PROGRAM Circuito_L7
VAR_INPUT
	Modo_Calibrar_L7: BOOL;
END_VAR
VAR
		fbBomba_L7 :Equipo_Motor_ATV320;
		ControlValv_ioLink_V1:ControlValv_ioLink;
		ControlValv_ioLink_V2: ControlValv_ioLink;
		ControlValv_ioLink_V3: ControlValv_ioLink;
		ControlValv_ioLink_V4: ControlValv_ioLink;
		Falla_L7_V1:BOOL;
		Falla_L7_V2:BOOL;
		Falla_L7_V3:BOOL;
		Falla_L7_V4:BOOL;
	Balanza_PU2_WT7: Balanza;
		dHS:DINT;
		TOF_calibradoIBC: TOF;
		PID_L7_SP:REAL;
		PID_L7_auto:BOOL;
		PID_L7_reset:BOOL;
		PID_L7_manual:REAL;
		PID_L7_bMuerta:REAL := 5;
		PID_L7_Kp:REAL := 0.1;
		PID_L7_Ti:REAL := 100;
		PID_L7_PV:REAL;
		Dosis_L7	:REAL;
		TiempoInyeccion_L7	:DINT;
		Peso	:REAL;
		Offset_L7:REAL;
		Inyeccion_L7:BOOL;
		Volumen_L7:REAL;
		Calculo_caudal_L7: Calculo_caudal;
		CorrecionCaudalxOffset_L7: CorrecionCaudalxOffset;
		tInyeccion: TON;
		Total :REAL;
		Totalant	:REAL;
		auxIniCal:BOOL;
		AuxVol:REAL;
		CA2_L7_V1_CmdA_Man :BOOL;
		CA2_L7_V4_CmdA_Man :BOOL;
		TDemoraInyectar: TON;
		SetDemoraInyeccion: REAL;
		Tiempo_seg_to_TIME_DemoraInyec: Tiempo_seg_to_TIME;
		AuxTDemoraInyec: TIME;
		PID_L7: FB_PID;
		Tiempo_TIME_to_seg_InyCal: Tiempo_TIME_to_seg;
		AuxInyCal:TIME;		
		IniTotalFT2:REAL;
		Auxconsumo:REAL;	
	ProductoAsociado: STRING;
	Lavagem_Circuito07: Lavagem;
	Calibracao_teste: Calibracao_V03;
END_VAR

VAR PERSISTENT
	UltimaCalibracao	:UDINT;	//Data e hora da ultima calibração
END_VAR
VAR // added by the converter: edge detectors and wires of the graphical bodies
    _w1, _w2, _w3, _w4, _w5, _w6, _w7, _w8, _w9, _w10, _w11, _w12, _w13 : BOOL;
    _ft1 : F_TRIG;
    _rt1, _rt2 : R_TRIG;
END_VAR

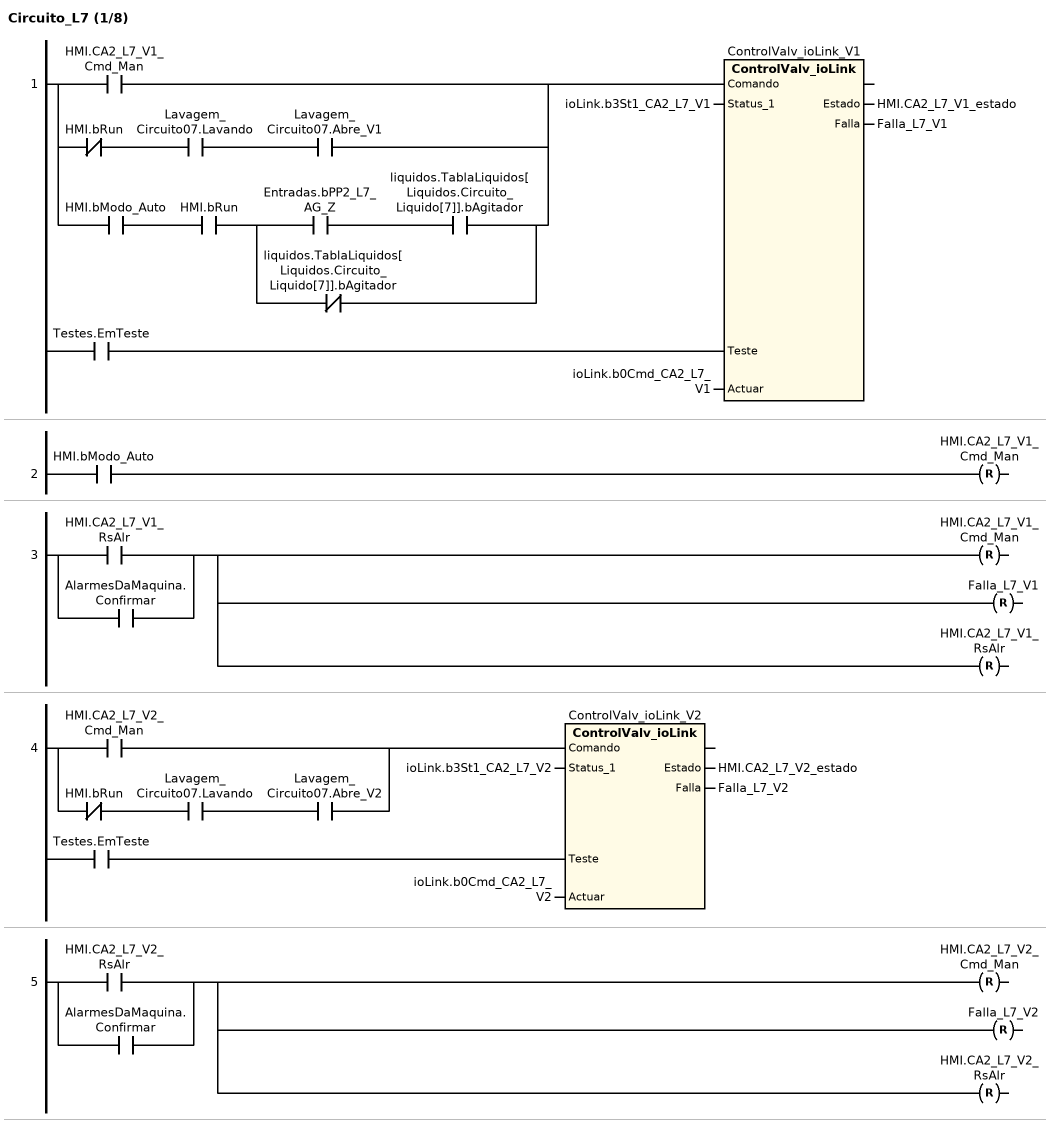
// NETWORK 1
ControlValv_ioLink_V1(
    Comando := HMI.CA2_L7_V1_Cmd_Man OR NOT HMI.bRun AND Lavagem_Circuito07.Lavando AND Lavagem_Circuito07.Abre_V1 OR HMI.bModo_Auto AND HMI.bRun AND (Entradas.bPP2_L7_AG_Z AND (liquidos.TablaLiquidos[Liquidos.Circuito_Liquido[7]].bAgitador) OR NOT (liquidos.TablaLiquidos[Liquidos.Circuito_Liquido[7]].bAgitador)),
    Status_1 := ioLink.b3St1_CA2_L7_V1,
    Teste := Testes.EmTeste,
    Actuar := ioLink.b0Cmd_CA2_L7_V1,
    Estado => HMI.CA2_L7_V1_estado,
    Falla => Falla_L7_V1); // ControlValv_ioLink

// NETWORK 2
HMI.CA2_L7_V1_Cmd_Man R= HMI.bModo_Auto;

// NETWORK 3
_w1 := HMI.CA2_L7_V1_RsAlr OR AlarmesDaMaquina.Confirmar;
HMI.CA2_L7_V1_Cmd_Man R= _w1;
Falla_L7_V1 R= _w1;
HMI.CA2_L7_V1_RsAlr R= _w1;

// NETWORK 4
ControlValv_ioLink_V2(
    Comando := HMI.CA2_L7_V2_Cmd_Man OR NOT HMI.bRun AND Lavagem_Circuito07.Lavando AND Lavagem_Circuito07.Abre_V2,
    Status_1 := ioLink.b3St1_CA2_L7_V2,
    Teste := Testes.EmTeste,
    Actuar := ioLink.b0Cmd_CA2_L7_V2,
    Estado => HMI.CA2_L7_V2_estado,
    Falla => Falla_L7_V2); // ControlValv_ioLink

// NETWORK 5
_w2 := HMI.CA2_L7_V2_RsAlr OR AlarmesDaMaquina.Confirmar;
HMI.CA2_L7_V2_Cmd_Man R= _w2;
Falla_L7_V2 R= _w2;
HMI.CA2_L7_V2_RsAlr R= _w2;

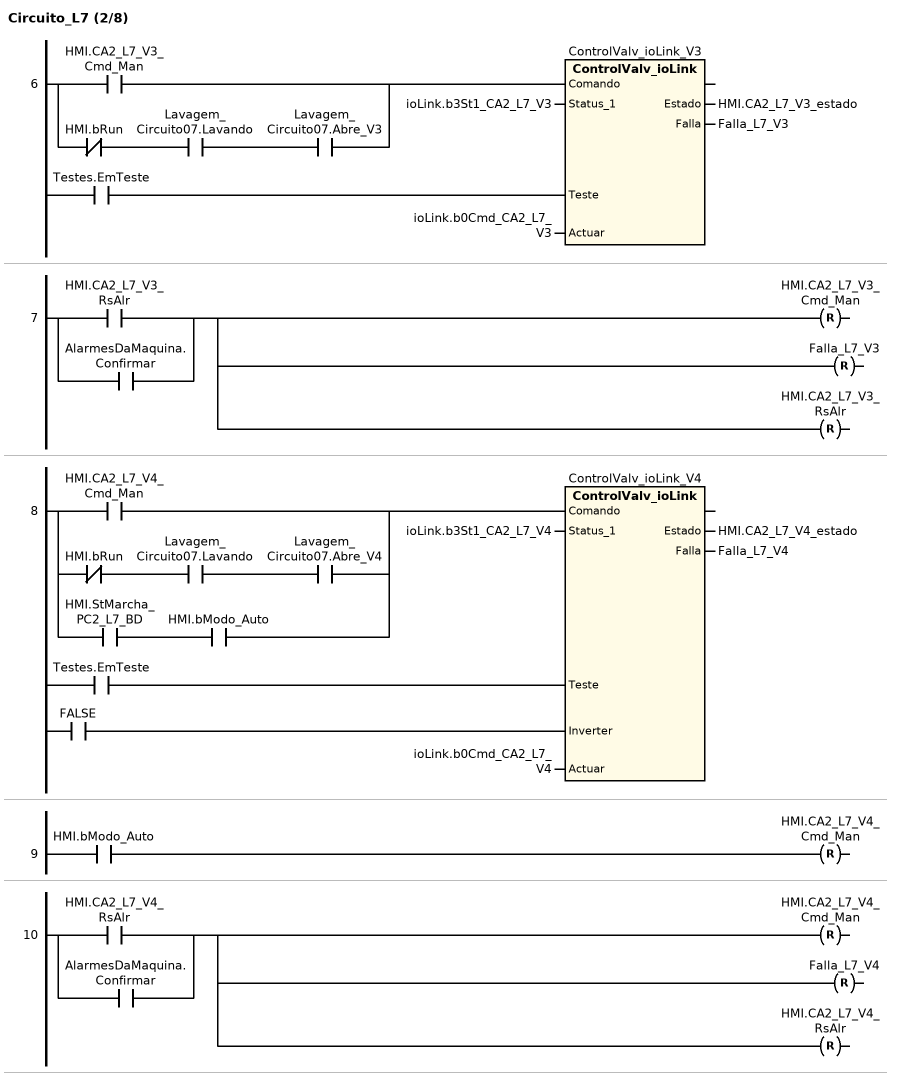
// NETWORK 6
ControlValv_ioLink_V3(
    Comando := HMI.CA2_L7_V3_Cmd_Man OR NOT HMI.bRun AND Lavagem_Circuito07.Lavando AND Lavagem_Circuito07.Abre_V3,
    Status_1 := ioLink.b3St1_CA2_L7_V3,
    Teste := Testes.EmTeste,
    Actuar := ioLink.b0Cmd_CA2_L7_V3,
    Estado => HMI.CA2_L7_V3_estado,
    Falla => Falla_L7_V3); // ControlValv_ioLink

// NETWORK 7
_w3 := HMI.CA2_L7_V3_RsAlr OR AlarmesDaMaquina.Confirmar;
HMI.CA2_L7_V3_Cmd_Man R= _w3;
Falla_L7_V3 R= _w3;
HMI.CA2_L7_V3_RsAlr R= _w3;

// NETWORK 8
ControlValv_ioLink_V4(
    Comando := HMI.CA2_L7_V4_Cmd_Man OR NOT HMI.bRun AND Lavagem_Circuito07.Lavando AND Lavagem_Circuito07.Abre_V4 OR HMI.StMarcha_PC2_L7_BD AND HMI.bModo_Auto,
    Status_1 := ioLink.b3St1_CA2_L7_V4,
    Teste := Testes.EmTeste,
    Inverter := FALSE,
    Actuar := ioLink.b0Cmd_CA2_L7_V4,
    Estado => HMI.CA2_L7_V4_estado,
    Falla => Falla_L7_V4); // ControlValv_ioLink

// NETWORK 9
HMI.CA2_L7_V4_Cmd_Man R= HMI.bModo_Auto;

// NETWORK 10
_w4 := HMI.CA2_L7_V4_RsAlr OR AlarmesDaMaquina.Confirmar;
HMI.CA2_L7_V4_Cmd_Man R= _w4;
Falla_L7_V4 R= _w4;
HMI.CA2_L7_V4_RsAlr R= _w4;

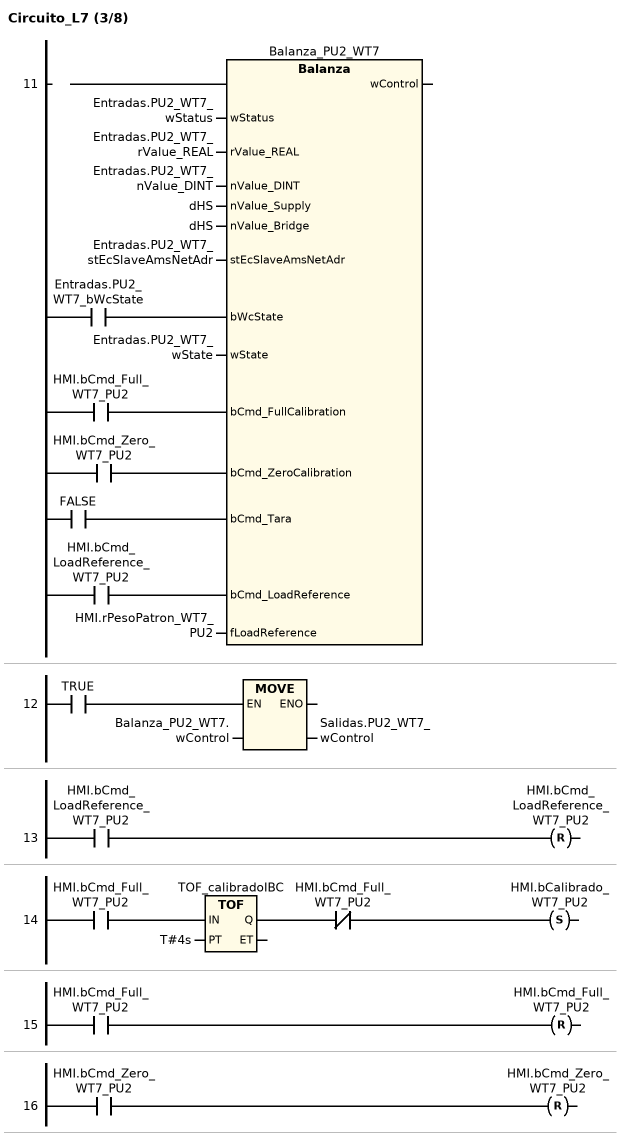
// NETWORK 11
Balanza_PU2_WT7(
    wStatus := Entradas.PU2_WT7_wStatus,
    rValue_REAL := Entradas.PU2_WT7_rValue_REAL,
    nValue_DINT := Entradas.PU2_WT7_nValue_DINT,
    nValue_Supply := dHS,
    nValue_Bridge := dHS,
    stEcSlaveAmsNetAdr := Entradas.PU2_WT7_stEcSlaveAmsNetAdr,
    bWcState := Entradas.PU2_WT7_bWcState,
    wState := Entradas.PU2_WT7_wState,
    bCmd_FullCalibration := HMI.bCmd_Full_WT7_PU2,
    bCmd_ZeroCalibration := HMI.bCmd_Zero_WT7_PU2,
    bCmd_Tara := FALSE,
    bCmd_LoadReference := HMI.bCmd_LoadReference_WT7_PU2,
    fLoadReference := HMI.rPesoPatron_WT7_PU2); // Balanza

// NETWORK 12
Salidas.PU2_WT7_wControl := Balanza_PU2_WT7.wControl;

// NETWORK 13
HMI.bCmd_LoadReference_WT7_PU2 R= HMI.bCmd_LoadReference_WT7_PU2;

// NETWORK 14
TOF_calibradoIBC(IN := HMI.bCmd_Full_WT7_PU2, PT := T#4s); // TOF
HMI.bCalibrado_WT7_PU2 S= TOF_calibradoIBC.Q AND NOT HMI.bCmd_Full_WT7_PU2;

// NETWORK 15
HMI.bCmd_Full_WT7_PU2 R= HMI.bCmd_Full_WT7_PU2;

// NETWORK 16
HMI.bCmd_Zero_WT7_PU2 R= HMI.bCmd_Zero_WT7_PU2;

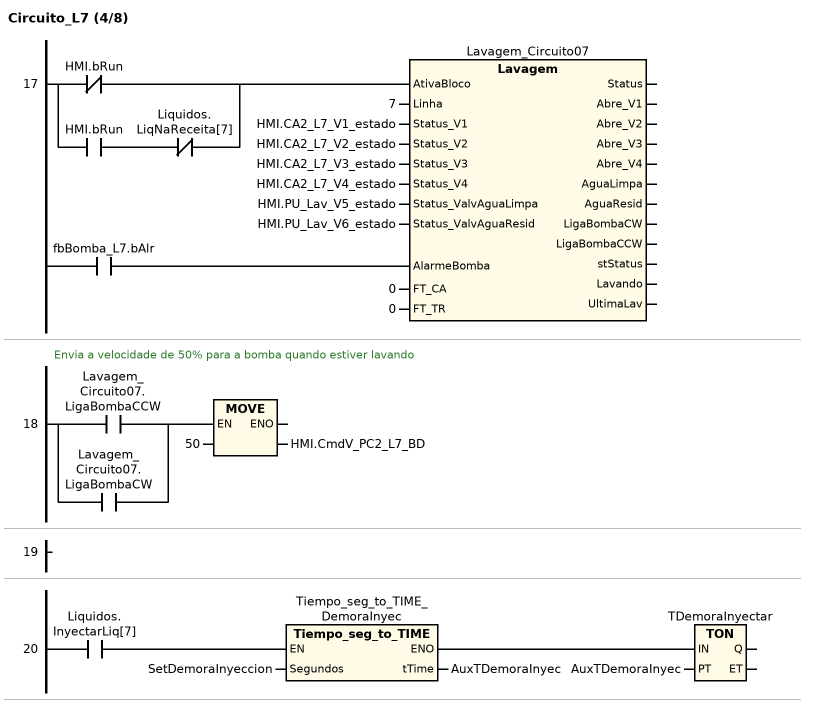
// NETWORK 17
Lavagem_Circuito07(
    AtivaBloco := NOT HMI.bRun OR HMI.bRun AND NOT Liquidos.LiqNaReceita[7],
    Linha := 7,
    Status_V1 := HMI.CA2_L7_V1_estado,
    Status_V2 := HMI.CA2_L7_V2_estado,
    Status_V3 := HMI.CA2_L7_V3_estado,
    Status_V4 := HMI.CA2_L7_V4_estado,
    Status_ValvAguaLimpa := HMI.PU_Lav_V5_estado,
    Status_ValvAguaResid := HMI.PU_Lav_V6_estado,
    AlarmeBomba := fbBomba_L7.bAlr,
    FT_CA := 0,
    FT_TR := 0); // Lavagem

// NETWORK 18
// Envia a velocidade de 50% para a bomba quando estiver lavando
IF Lavagem_Circuito07.LigaBombaCCW OR Lavagem_Circuito07.LigaBombaCW THEN HMI.CmdV_PC2_L7_BD := 50; END_IF

// NETWORK 19

// NETWORK 20
_w5 := Liquidos.InyectarLiq[7];
IF _w5 THEN
    Tiempo_seg_to_TIME_DemoraInyec(Segundos := SetDemoraInyeccion, tTime => AuxTDemoraInyec); // Tiempo_seg_to_TIME
END_IF
TDemoraInyectar(IN := _w5, PT := AuxTDemoraInyec); // TON

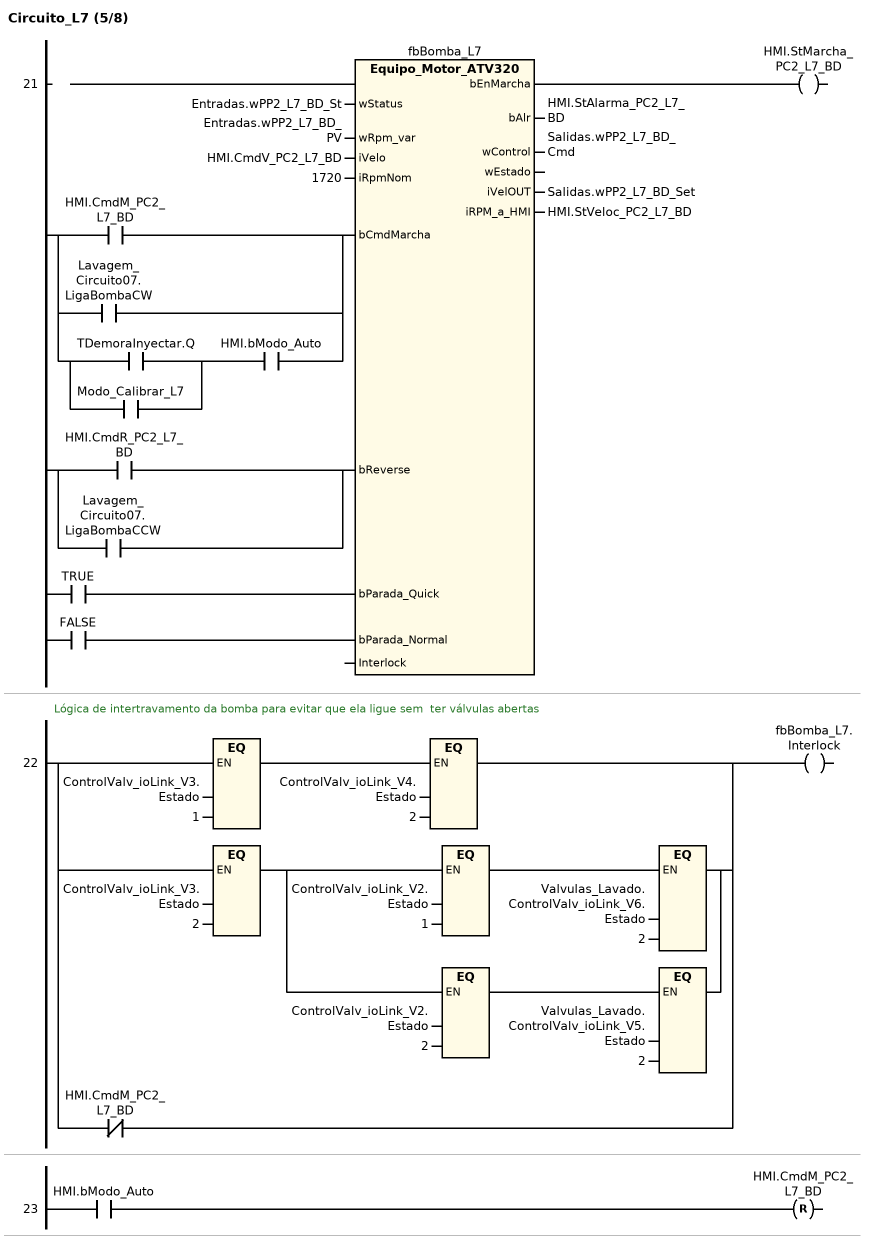
// NETWORK 21
fbBomba_L7(
    wStatus := Entradas.wPP2_L7_BD_St,
    wRpm_var := Entradas.wPP2_L7_BD_PV,
    iVelo := HMI.CmdV_PC2_L7_BD,
    iRpmNom := 1720,
    bCmdMarcha := HMI.CmdM_PC2_L7_BD OR Lavagem_Circuito07.LigaBombaCW OR (TDemoraInyectar.Q OR Modo_Calibrar_L7) AND HMI.bModo_Auto,
    bReverse := HMI.CmdR_PC2_L7_BD OR Lavagem_Circuito07.LigaBombaCCW,
    bParada_Quick := TRUE,
    bParada_Normal := FALSE,
    bAlr => HMI.StAlarma_PC2_L7_BD,
    wControl => Salidas.wPP2_L7_BD_Cmd,
    iVelOUT => Salidas.wPP2_L7_BD_Set,
    iRPM_a_HMI => HMI.StVeloc_PC2_L7_BD); // Equipo_Motor_ATV320
HMI.StMarcha_PC2_L7_BD := fbBomba_L7.bEnMarcha;

// NETWORK 22
// Lógica de intertravamento da bomba para evitar que ela ligue sem  ter válvulas abertas
_w6 := NOT HMI.CmdM_PC2_L7_BD;
IF NOT _w6 THEN
    _w7 := ControlValv_ioLink_V3.Estado = 2;
    _w6 := ControlValv_ioLink_V3.Estado = 1 AND ControlValv_ioLink_V4.Estado = 2 OR (_w7 AND ControlValv_ioLink_V2.Estado = 1 AND Valvulas_Lavado.ControlValv_ioLink_V6.Estado = 2 OR _w7 AND ControlValv_ioLink_V2.Estado = 2 AND Valvulas_Lavado.ControlValv_ioLink_V5.Estado = 2);
END_IF
fbBomba_L7.Interlock := _w6;

// NETWORK 23
HMI.CmdM_PC2_L7_BD R= HMI.bModo_Auto;

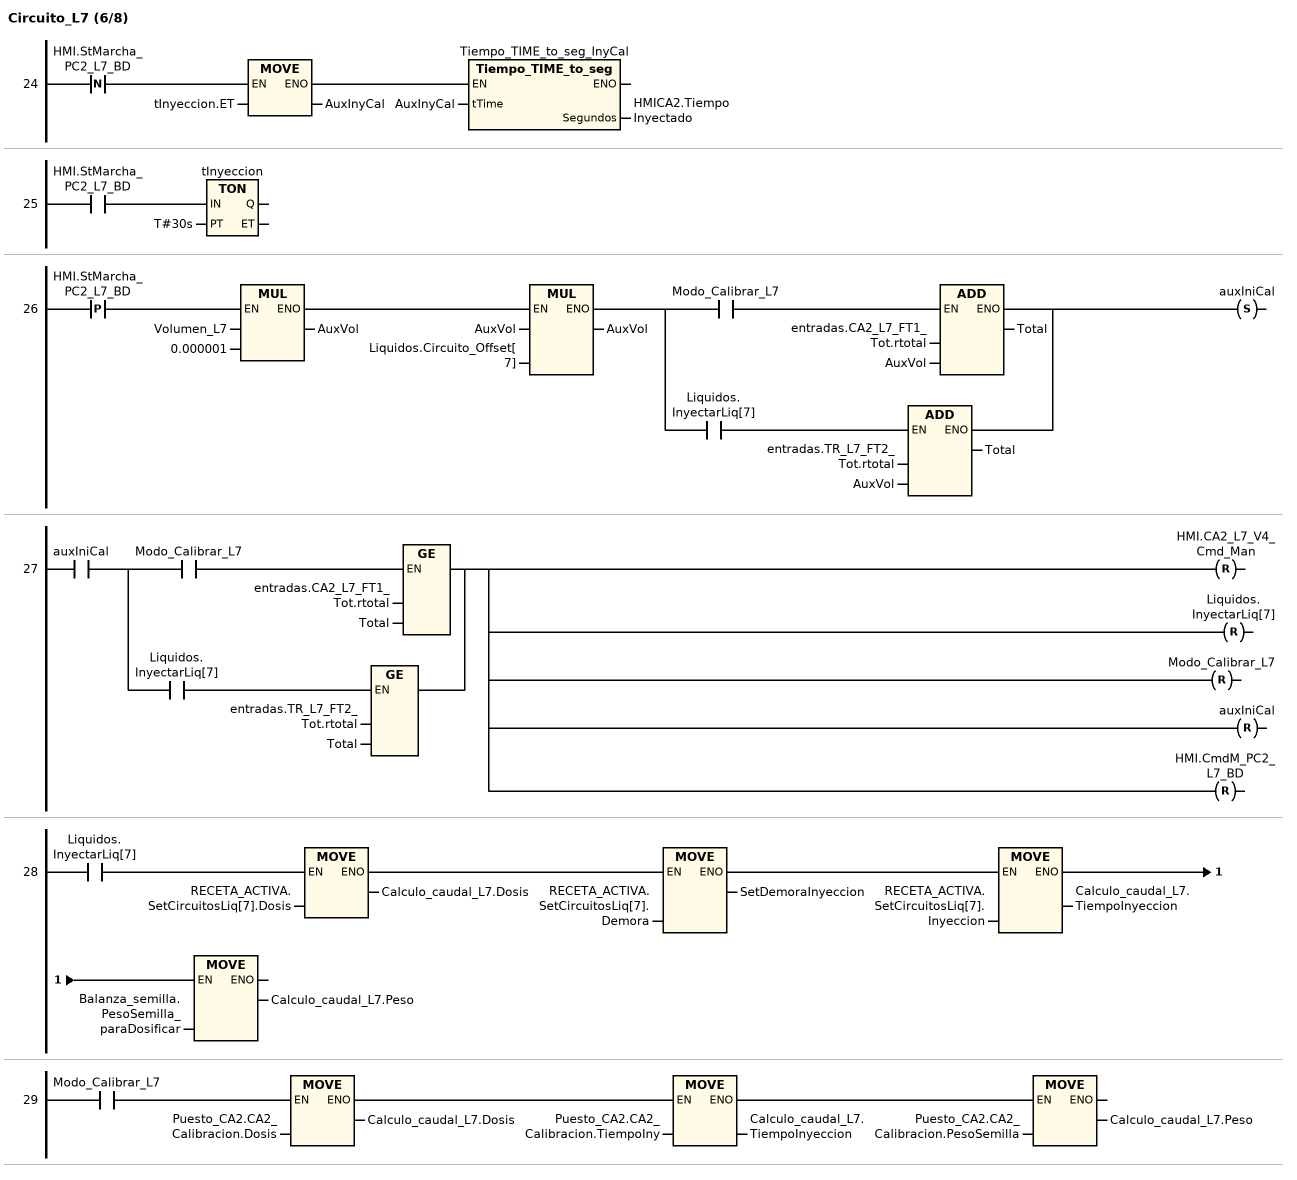
// NETWORK 24
_ft1(CLK := HMI.StMarcha_PC2_L7_BD);
_w8 := _ft1.Q;
IF _w8 THEN AuxInyCal := tInyeccion.ET; END_IF
IF _w8 THEN
    Tiempo_TIME_to_seg_InyCal(tTime := AuxInyCal, Segundos => HMICA2.TiempoInyectado); // Tiempo_TIME_to_seg
END_IF

// NETWORK 25
tInyeccion(IN := HMI.StMarcha_PC2_L7_BD, PT := T#30s); // TON

// NETWORK 26
_rt1(CLK := HMI.StMarcha_PC2_L7_BD);
_w9 := _rt1.Q;
IF _w9 THEN AuxVol := Volumen_L7 * 0.000001; END_IF
IF _w9 THEN AuxVol := AuxVol * Liquidos.Circuito_Offset[7]; END_IF
IF _w9 AND Modo_Calibrar_L7 THEN Total := entradas.CA2_L7_FT1_Tot.rtotal + AuxVol; END_IF
IF _w9 AND Liquidos.InyectarLiq[7] THEN Total := entradas.TR_L7_FT2_Tot.rtotal + AuxVol; END_IF
auxIniCal S= _w9 AND Modo_Calibrar_L7 OR _w9 AND Liquidos.InyectarLiq[7];

// NETWORK 27
_w10 := auxIniCal AND Modo_Calibrar_L7 AND entradas.CA2_L7_FT1_Tot.rtotal >= Total OR auxIniCal AND Liquidos.InyectarLiq[7] AND entradas.TR_L7_FT2_Tot.rtotal >= Total;
HMI.CA2_L7_V4_Cmd_Man R= _w10;
Liquidos.InyectarLiq[7] R= _w10;
Modo_Calibrar_L7 R= _w10;
auxIniCal R= _w10;
HMI.CmdM_PC2_L7_BD R= _w10;

// NETWORK 28
_w11 := Liquidos.InyectarLiq[7];
IF _w11 THEN Calculo_caudal_L7.Dosis := RECETA_ACTIVA.SetCircuitosLiq[7].Dosis; END_IF
IF _w11 THEN SetDemoraInyeccion := RECETA_ACTIVA.SetCircuitosLiq[7].Demora; END_IF
IF _w11 THEN Calculo_caudal_L7.TiempoInyeccion := RECETA_ACTIVA.SetCircuitosLiq[7].Inyeccion; END_IF
IF _w11 THEN Calculo_caudal_L7.Peso := Balanza_semilla.PesoSemilla_paraDosificar; END_IF

// NETWORK 29
_w12 := Modo_Calibrar_L7;
IF _w12 THEN Calculo_caudal_L7.Dosis := Puesto_CA2.CA2_Calibracion.Dosis; END_IF
IF _w12 THEN Calculo_caudal_L7.TiempoInyeccion := Puesto_CA2.CA2_Calibracion.TiempoIny; END_IF
IF _w12 THEN Calculo_caudal_L7.Peso := Puesto_CA2.CA2_Calibracion.PesoSemilla; END_IF

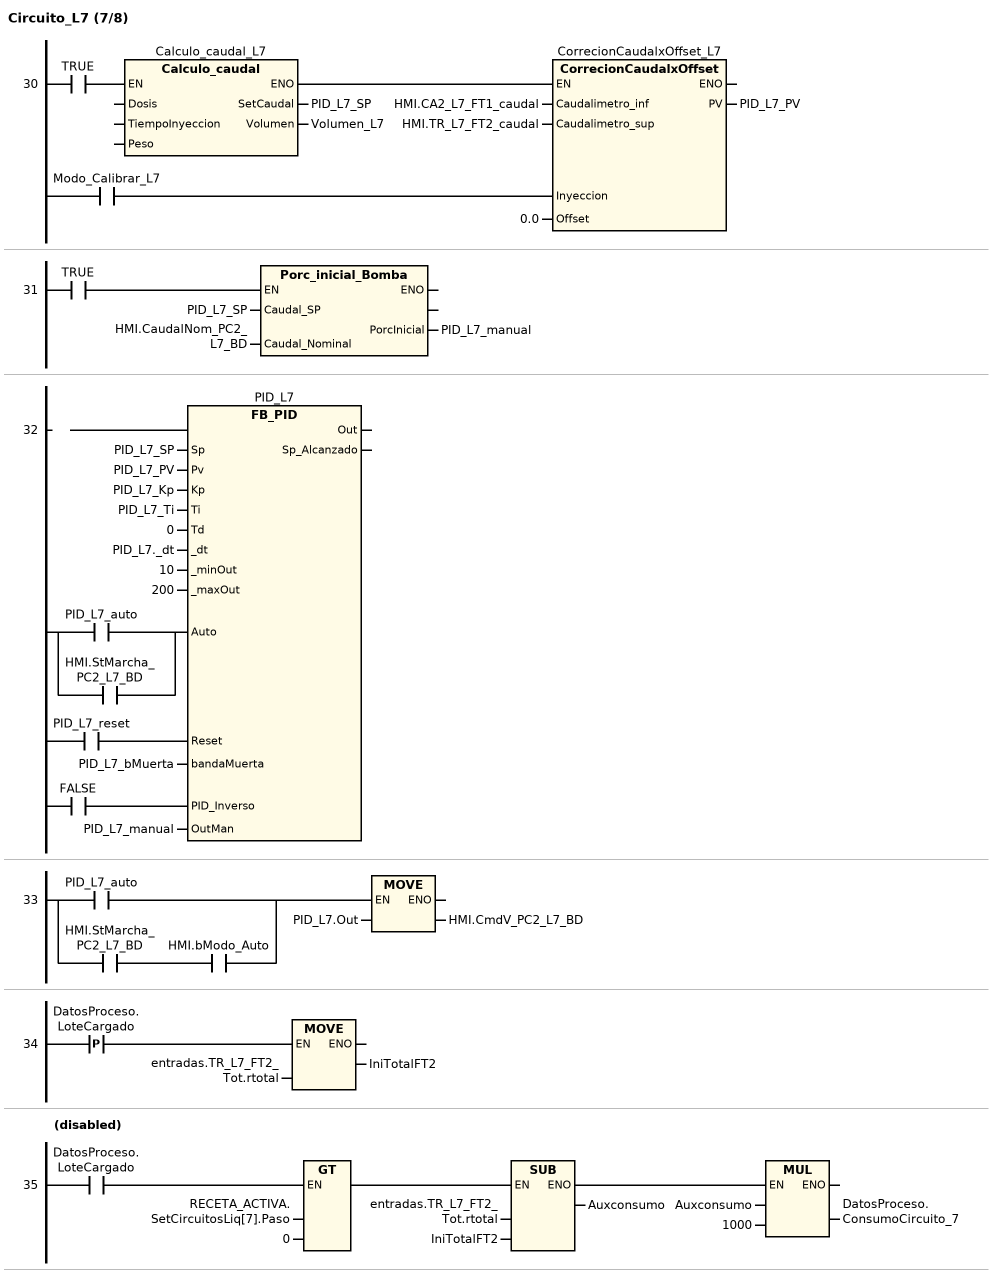
// NETWORK 30
Calculo_caudal_L7(SetCaudal => PID_L7_SP, Volumen => Volumen_L7); // Calculo_caudal
CorrecionCaudalxOffset_L7(
    Caudalimetro_inf := HMI.CA2_L7_FT1_caudal,
    Caudalimetro_sup := HMI.TR_L7_FT2_caudal,
    Inyeccion := Modo_Calibrar_L7,
    Offset := 0.0,
    PV => PID_L7_PV); // CorrecionCaudalxOffset

// NETWORK 31
Porc_inicial_Bomba(Caudal_SP := PID_L7_SP, Caudal_Nominal := HMI.CaudalNom_PC2_L7_BD, PorcInicial => PID_L7_manual);

// NETWORK 32
PID_L7(
    Sp := PID_L7_SP,
    Pv := PID_L7_PV,
    Kp := PID_L7_Kp,
    Ti := PID_L7_Ti,
    Td := 0,
    _dt := PID_L7._dt,
    _minOut := 10,
    _maxOut := 200,
    Auto := PID_L7_auto OR HMI.StMarcha_PC2_L7_BD,
    Reset := PID_L7_reset,
    bandaMuerta := PID_L7_bMuerta,
    PID_Inverso := FALSE,
    OutMan := PID_L7_manual); // FB_PID

// NETWORK 33
IF PID_L7_auto OR HMI.StMarcha_PC2_L7_BD AND HMI.bModo_Auto THEN HMI.CmdV_PC2_L7_BD := PID_L7.Out; END_IF

// NETWORK 34
_rt2(CLK := DatosProceso.LoteCargado);
IF _rt2.Q THEN IniTotalFT2 := entradas.TR_L7_FT2_Tot.rtotal; END_IF

// NETWORK 35 (disabled)
// _w13 := DatosProceso.LoteCargado AND RECETA_ACTIVA.SetCircuitosLiq[7].Paso > 0;
// IF _w13 THEN Auxconsumo := entradas.TR_L7_FT2_Tot.rtotal - IniTotalFT2; END_IF
// IF _w13 THEN DatosProceso.ConsumoCircuito_7 := Auxconsumo * 1000; END_IF

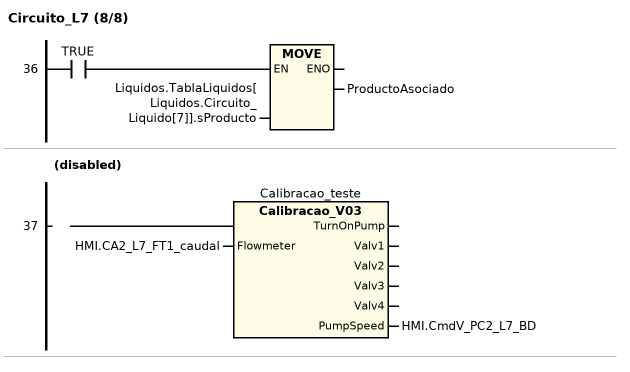
// NETWORK 36
ProductoAsociado := Liquidos.TablaLiquidos[Liquidos.Circuito_Liquido[7]].sProducto;

// NETWORK 37 (disabled)
// Calibracao_teste(Flowmeter := HMI.CA2_L7_FT1_caudal, PumpSpeed => HMI.CmdV_PC2_L7_BD); // Calibracao_V03

END_PROGRAM

(* stored: Version 1.1.0.1, ProductVersion 3.1.4024.14
   POU Circuito_L7: Id {a76ea28e-4919-4c84-b82d-2e33c4595a07}, SpecialFunc None *)
